INTERFACE I_MoveAbsolute EXTENDS I_StatusEx

METHOD ClearStatus
VAR_INPUT
END_VAR
END_METHOD

METHOD MoveAbsolute
VAR_INPUT
    Position	: LREAL;
    Velocity	: LREAL;
    Acceleration	: LREAL := 0.0;
    Deceleration	: LREAL := 0.0;
    Jerk	: LREAL := 0.0;
    BufferMode	: MC_BufferMode := MC_BufferMode.MC_Aborting;
END_VAR
END_METHOD

END_INTERFACE

(* stored: Version 1.1.0.1
   Itf I_MoveAbsolute: Id {7b52c23d-d549-4d14-b715-d0e842580738}
   Method ClearStatus: Id {6a802a6a-3cf0-40e8-a1d5-b17dc4cbc118}
   Method MoveAbsolute: Id {6ca50ed1-00a4-4a5f-9fc0-b477fbaad08d} *)
